(* IEC 61131-3 sources: pic32mz-nolib/stfile, 4 files *)

(* ---- st_file.st ---- *)
PROGRAM program0
  VAR
    bstart AT %IX0.15 : BOOL;
    bstop AT %IX0.14 : BOOL;
    led AT %QX0.15 : BOOL;
    var_byte AT %MB0 : SINT;
    var_long AT %ML0 : ULINT;
  END_VAR

  led := NOT(bstop) AND (bstart OR led);
END_PROGRAM

CONFIGURATION Config0

  RESOURCE Res0 ON PLC
    TASK task0(INTERVAL := T#1ms,PRIORITY := 0);
    PROGRAM instance0 WITH task0 : program0;
  END_RESOURCE
END_CONFIGURATION

(* ---- st_file_0.st ---- *)
PROGRAM moreadvance
  VAR
    m_run AT %IX0.0 : BOOL;
  END_VAR
  VAR
    timvalue : TIME := T#1000ms;
  END_VAR
  VAR
    m_stop AT %IX0.1 : BOOL;
    m_dir AT %IX0.2 : BOOL;
    m_fw AT %QX0.0 : BOOL;
    m_bw AT %QX0.1 : BOOL;
    m_led AT %QX0.2 : BOOL;
  END_VAR
  VAR
    m_state : BOOL;
    TON0 : TON;
    TON1 : TON;
  END_VAR
  VAR_INPUT
    test : BOOL;
  END_VAR
  VAR
    GT20_OUT : BOOL;
  END_VAR

  m_state := NOT(m_stop) AND (m_run OR m_state);
  TON0(IN := m_state AND m_dir, PT := timvalue);
  m_fw := TON0.Q;
  TON1(IN := m_state AND NOT(m_dir), PT := T#1000ms);
  m_bw := TON1.Q;
  GT20_OUT := GT(TON0.ET, TON1.ET);
  m_led := GT20_OUT;
END_PROGRAM

CONFIGURATION Config0

  RESOURCE Res0 ON PLC
    VAR_GLOBAL
      version : DINT;
    END_VAR
    TASK task0(INTERVAL := T#20ms,PRIORITY := 0);
    PROGRAM instance0 WITH task0 : moreadvance;
  END_RESOURCE
END_CONFIGURATION

(* ---- st_file_1.st ---- *)
PROGRAM program0
  VAR
    count AT %IX0.0 : BOOL;
    r_count AT %IX0.1 : BOOL;
    count_reach AT %QX0.0 : BOOL;
  END_VAR
  VAR
    curr_count : INT;
    CTU0 : CTU;
    R_TRIG1 : R_TRIG;
    R_TRIG2 : R_TRIG;
    R_TRIG3 : R_TRIG;
  END_VAR

  R_TRIG1(CLK := count);
  R_TRIG2(CLK := R_TRIG1.Q);
  R_TRIG3(CLK := r_count);
  CTU0(CU := R_TRIG2.Q, R := R_TRIG3.Q, PV := 5);
  count_reach := CTU0.Q;
  curr_count := CTU0.CV;
END_PROGRAM

CONFIGURATION Config0

  RESOURCE Res0 ON PLC
    TASK task0(INTERVAL := T#20ms,PRIORITY := 0);
    PROGRAM instance0 WITH task0 : program0;
  END_RESOURCE
END_CONFIGURATION

(* ---- st_file_2.st ---- *)
PROGRAM program0
  VAR
    tmpreset AT %MD0 : REAL := 3.0;
    poweron AT %IX0.0 : BOOL;
    lamp AT %QX0.1 : BOOL;
  END_VAR
  VAR
    TOF0 : TOF;
    REAL_TO_TIME8_OUT : TIME;
  END_VAR

  REAL_TO_TIME8_OUT := REAL_TO_TIME(tmpreset);
  TOF0(IN := poweron, PT := REAL_TO_TIME8_OUT);
  lamp := TOF0.Q;
END_PROGRAM

CONFIGURATION Config0

  RESOURCE Res0 ON PLC
    TASK task0(INTERVAL := T#1ms,PRIORITY := 0);
    PROGRAM instance0 WITH task0 : program0;
  END_RESOURCE
END_CONFIGURATION
